{attribute 'qualified_only'}
{attribute 'strict'}
{attribute 'to_string'}
TYPE
	eFTPState :(
		Disconnected := 0,	
		Connecting := 1,      
		Downloading := 2,      
		Success := 3,    
		Failure := 4
	);
END_TYPE

(* stored: Version 1.1.0.1, ProductVersion 3.1.4026.18
   DUT eFTPState: Id {fc3cc688-6907-4290-83b6-f3902dee2262} *)
